FUNCTION_BLOCK FB_Loadcell IMPLEMENTS I_LoadCell
VAR_INPUT
	idDevice					: INT;// 1: mettler		,2: Laumas
END_VAR
VAR_OUTPUT
	Error						: BOOL;
END_VAR
VAR
	ondinh						: BOOL;
	fbInterface					: FB_Interface_EtherCat;
	nErrID						: INT;	
END_VAR

fbInterface(idDevice := idDevice,Error => Error);

PROPERTY fActWeight : REAL
GET
fActWeight := fbInterface.fActWeight;
END_GET
END_PROPERTY

METHOD NetMode : BOOL
VAR_INPUT
END_VAR
fbInterface.NetMode();
END_METHOD

METHOD Set_Zero : BOOL
VAR_INPUT
END_VAR
fbInterface.Set_Zero();
END_METHOD

PROPERTY Status : REAL;
GET
Status := fbInterface.Status;
END_GET
END_PROPERTY

END_FUNCTION_BLOCK

(* stored: Version 1.1.0.1, ProductVersion 3.1.4024.12
   POU FB_Loadcell: Id {eac700fd-516e-4b65-9e0d-da734dceffb1}, SpecialFunc None
   Property fActWeight: Id {39c3a08a-5660-407b-8ef5-42f965139c39}
   Get Get: Id {173c3f43-b986-44d7-85a7-e573e4ad3b09}
   Method NetMode: Id {46589393-1d53-4dda-b644-734e3962c876}
   Method Set_Zero: Id {ec782a9a-cbf8-48fe-bf1c-ccc1593dd634}
   Property Status: Id {cbb2df3e-a8fb-4d7c-9ed5-b965ae25b583}
   Get Get: Id {092ba072-b294-46d9-8862-dc1c640858c4} *)
